// TIA Portal V17 export
// export: Created 2023-04-05T15:02:24.3314594Z, ExportSetting WithDefaults, DisplayName Totally Integrated Automation Portal, DisplayVersion V17 Update 4, DisplayName TIA Portal Openness, DisplayVersion V17 Update 4, DisplayName TIA Portal Version Control Interface, DisplayVersion V17, DisplayName STEP 7 Professional, DisplayVersion V17 Update 4, DisplayName STEP 7 Safety, DisplayVersion V17, DisplayName WinCC Professional, DisplayVersion V17 Update 4
FUNCTION_BLOCK "Main_Safety_RTG1"   // FB501, F_LAD
{ S7_Optimized_Access := 'TRUE' }
VERSION : 0.1
// stored: AutoNumber false, IsIECCheckEnabled false, UDAEnableTagReadback false
BEGIN

REGION Network 1: Receive data from Core - new
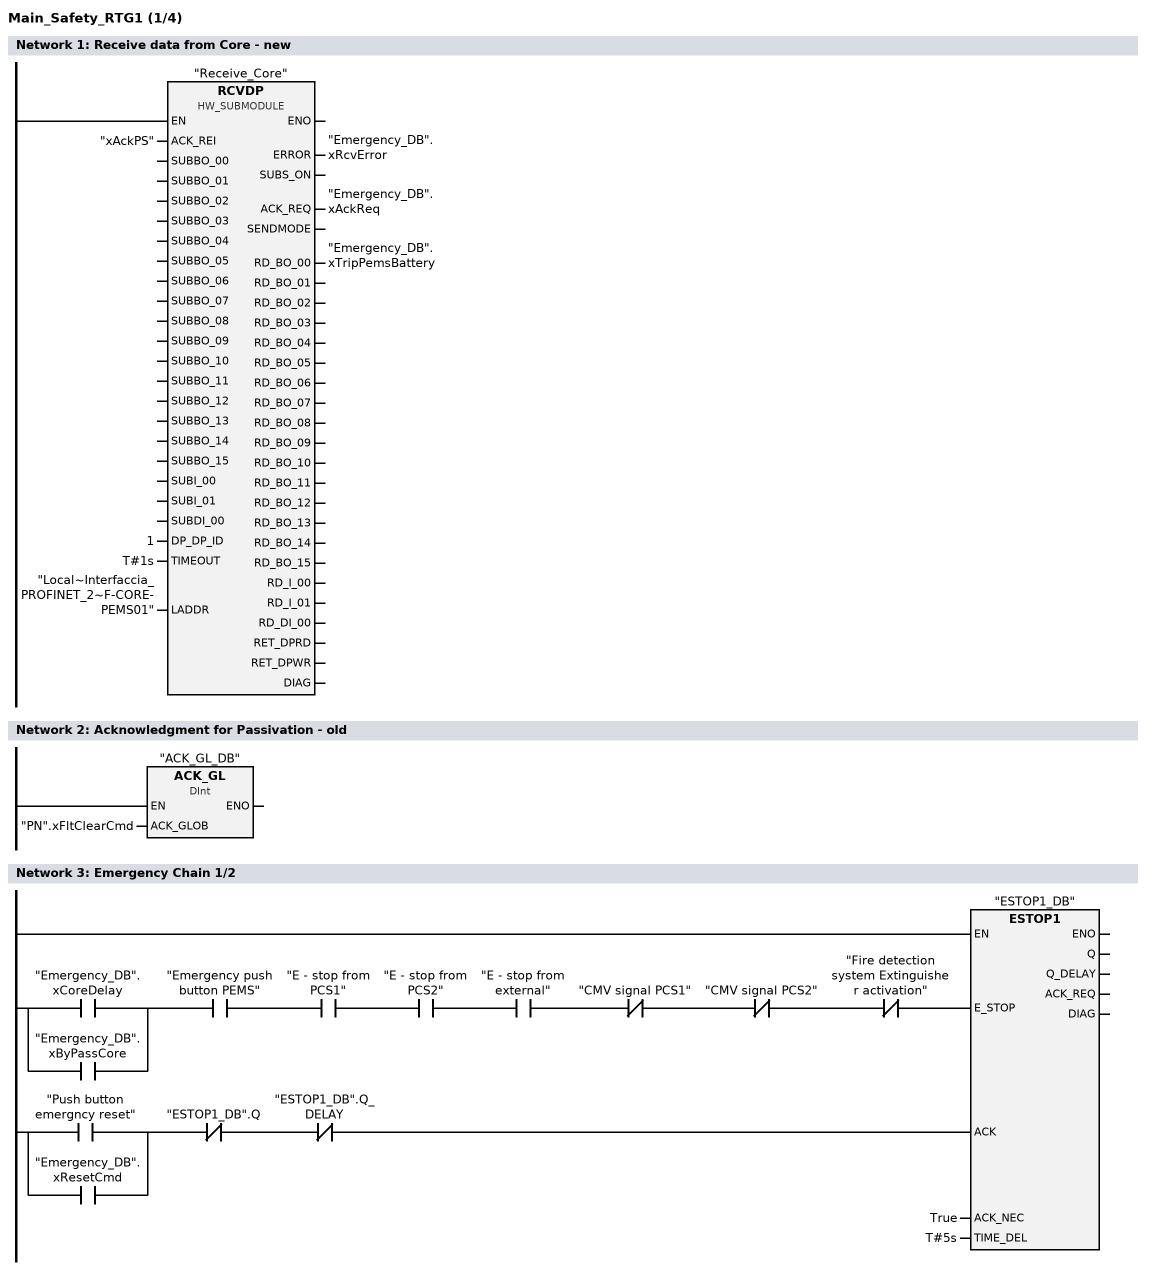
   RUNG wire#powerrail
      { S7_Templates := "laddr_type := HW_SUBMODULE" } "Receive_Core".RCVDP(ACK_REI := "xAckPS", SUBBO_00 :=, SUBBO_01 :=, SUBBO_02 :=, SUBBO_03 :=, SUBBO_04 :=, SUBBO_05 :=, SUBBO_06 :=, SUBBO_07 :=, SUBBO_08 :=, SUBBO_09 :=, SUBBO_10 :=, SUBBO_11 :=, SUBBO_12 :=, SUBBO_13 :=, SUBBO_14 :=, SUBBO_15 :=, SUBI_00 :=, SUBI_01 :=, SUBDI_00 :=, DP_DP_ID := 1, TIMEOUT := T#1s, LADDR := "Local~Interfaccia_PROFINET_2~F-CORE-PEMS01", ERROR => "Emergency_DB".xRcvError, SUBS_ON =>, ACK_REQ => "Emergency_DB".xAckReq, SENDMODE =>, RD_BO_00 => "Emergency_DB".xTripPemsBattery, RD_BO_01 =>, RD_BO_02 =>, RD_BO_03 =>, RD_BO_04 =>, RD_BO_05 =>, RD_BO_06 =>, RD_BO_07 =>, RD_BO_08 =>, RD_BO_09 =>, RD_BO_10 =>, RD_BO_11 =>, RD_BO_12 =>, RD_BO_13 =>, RD_BO_14 =>, RD_BO_15 =>, RD_I_00 =>, RD_I_01 =>, RD_DI_00 =>, RET_DPRD =>, RET_DPWR =>, DIAG =>)
   END_RUNG
   // the same network as SCL:
   "Receive_Core"(ACK_REI := "xAckPS",   // RCVDP
                  DP_DP_ID := 1,
                  TIMEOUT := T#1s,
                  LADDR := "Local~Interfaccia_PROFINET_2~F-CORE-PEMS01",
                  ERROR => "Emergency_DB".xRcvError,
                  ACK_REQ => "Emergency_DB".xAckReq,
                  RD_BO_00 => "Emergency_DB".xTripPemsBattery);
END_REGION

REGION Network 2: Acknowledgment for Passivation - old
   RUNG wire#powerrail
      { S7_Templates := "codedbool_type := DInt" } "ACK_GL_DB".ACK_GL(ACK_GLOB := "PN".xFltClearCmd)
   END_RUNG
   // the same network as SCL:
   "ACK_GL_DB"(ACK_GLOB := "PN".xFltClearCmd);   // ACK_GL
END_REGION

REGION Network 3: Emergency Chain 1/2
   RUNG wire#powerrail
      "ESTOP1_DB".ESTOP1(E_STOP := wire#w2, ACK := wire#w4, ACK_NEC := True, TIME_DEL := T#5s, Q =>, Q_DELAY =>, ACK_REQ =>, DIAG =>)
   END_RUNG
   RUNG wire#powerrail
      Contact( "Emergency_DB".xCoreDelay )
      wire#w1
      Contact( "Emergency push button PEMS" )
      Contact( "E - stop from PCS1" )
      Contact( "E - stop from PCS2" )
      Contact( "E - stop from external" )
      I_Contact( "CMV signal PCS1" )
      I_Contact( "CMV signal PCS2" )
      I_Contact( "Fire detection system Extinguisher activation" )
   END_RUNG wire#w2
   RUNG wire#powerrail
      Contact( "Emergency_DB".xByPassCore )
   END_RUNG wire#w1
   RUNG wire#powerrail
      Contact( "Push button emergncy reset" )
      wire#w3
      I_Contact( "ESTOP1_DB".Q )
      I_Contact( "ESTOP1_DB".Q_DELAY )
   END_RUNG wire#w4
   RUNG wire#powerrail
      Contact( "Emergency_DB".xResetCmd )
   END_RUNG wire#w3
   // the same network as SCL:
   "ESTOP1_DB"(E_STOP := ("Emergency_DB".xCoreDelay OR "Emergency_DB".xByPassCore) AND "Emergency push button PEMS" AND "E - stop from PCS1" AND "E - stop from PCS2" AND "E - stop from external" AND NOT "CMV signal PCS1" AND NOT "CMV signal PCS2" AND NOT "Fire detection system Extinguisher activation",   // ESTOP1
               ACK := ("Push button emergncy reset" OR "Emergency_DB".xResetCmd) AND NOT "ESTOP1_DB".Q AND NOT "ESTOP1_DB".Q_DELAY,
               ACK_NEC := True,
               TIME_DEL := T#5s);
END_REGION

REGION Network 4: Emergency shunt opening release RESET
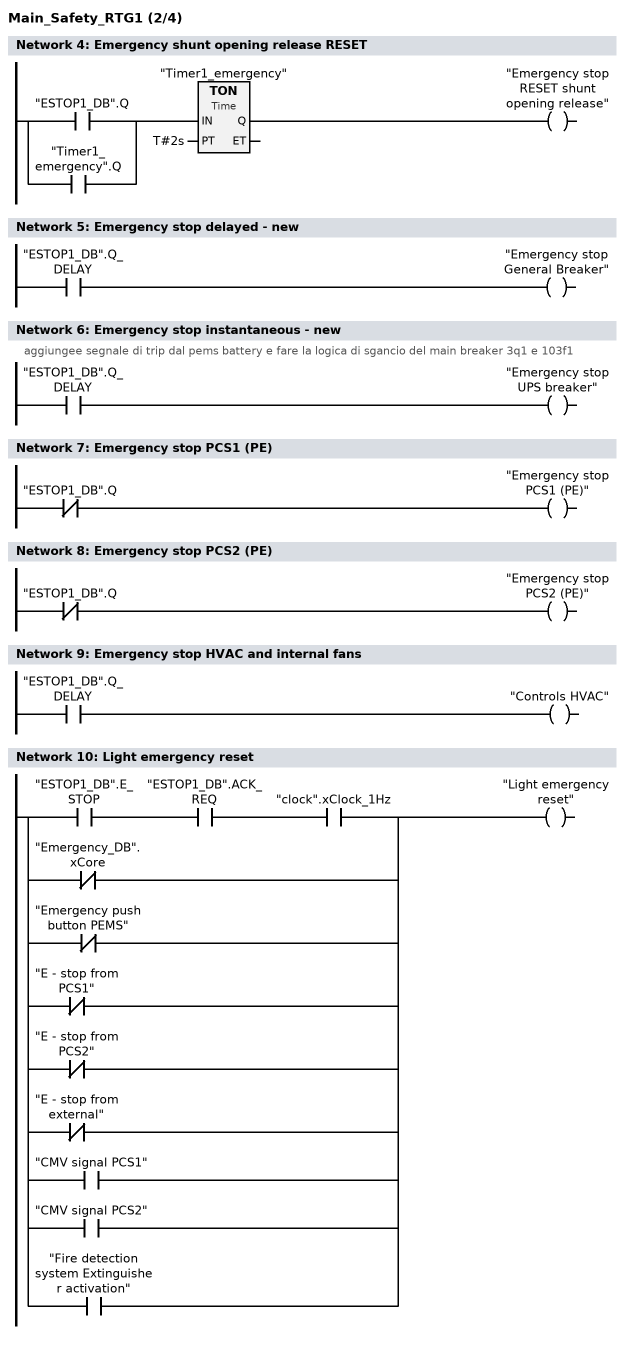
   RUNG wire#powerrail
      Contact( "ESTOP1_DB".Q )
      wire#w1
      { S7_Templates := "[time_type := Time, codedbool_type := DInt]" } "Timer1_emergency".TON(pt := T#2s, et =>)
      Coil( "Emergency stop RESET shunt opening release" )
   END_RUNG
   RUNG wire#powerrail
      Contact( "Timer1_emergency".Q )
   END_RUNG wire#w1
   // the same network as SCL:
   "Timer1_emergency".TON(IN := "ESTOP1_DB".Q OR "Timer1_emergency".Q, PT := T#2s);
   "Emergency stop RESET shunt opening release" := "Timer1_emergency".Q;
END_REGION

REGION Network 5: Emergency stop delayed - new
   RUNG wire#powerrail
      Contact( "ESTOP1_DB".Q_DELAY )
      Coil( "Emergency stop General Breaker" )
   END_RUNG
   // the same network as SCL:
   "Emergency stop General Breaker" := "ESTOP1_DB".Q_DELAY;
END_REGION

REGION Network 6: Emergency stop instantaneous - new
   // aggiungee segnale di trip dal pems battery e fare la logica di sgancio del main breaker 3q1 e 103f1
   RUNG wire#powerrail
      Contact( "ESTOP1_DB".Q_DELAY )
      Coil( "Emergency stop UPS breaker" )
   END_RUNG
   // the same network as SCL:
   "Emergency stop UPS breaker" := "ESTOP1_DB".Q_DELAY;
END_REGION

REGION Network 7: Emergency stop PCS1 (PE)
   RUNG wire#powerrail
      I_Contact( "ESTOP1_DB".Q )
      Coil( "Emergency stop PCS1 (PE)" )
   END_RUNG
   // the same network as SCL:
   "Emergency stop PCS1 (PE)" := NOT "ESTOP1_DB".Q;
END_REGION

REGION Network 8: Emergency stop PCS2 (PE)
   RUNG wire#powerrail
      I_Contact( "ESTOP1_DB".Q )
      Coil( "Emergency stop PCS2 (PE)" )
   END_RUNG
   // the same network as SCL:
   "Emergency stop PCS2 (PE)" := NOT "ESTOP1_DB".Q;
END_REGION

REGION Network 9: Emergency stop HVAC and internal fans
   RUNG wire#powerrail
      Contact( "ESTOP1_DB".Q_DELAY )
      Coil( "Controls HVAC" )
   END_RUNG
   // the same network as SCL:
   "Controls HVAC" := "ESTOP1_DB".Q_DELAY;
END_REGION

REGION Network 10: Light emergency reset
   RUNG wire#powerrail
      Contact( "ESTOP1_DB".E_STOP )
      Contact( "ESTOP1_DB".ACK_REQ )
      Contact( "clock".xClock_1Hz )
      wire#w1
      Coil( "Light emergency reset" )
   END_RUNG
   RUNG wire#powerrail
      I_Contact( "Emergency_DB".xCore )
   END_RUNG wire#w1
   RUNG wire#powerrail
      I_Contact( "Emergency push button PEMS" )
   END_RUNG wire#w1
   RUNG wire#powerrail
      I_Contact( "E - stop from PCS1" )
   END_RUNG wire#w1
   RUNG wire#powerrail
      I_Contact( "E - stop from PCS2" )
   END_RUNG wire#w1
   RUNG wire#powerrail
      I_Contact( "E - stop from external" )
   END_RUNG wire#w1
   RUNG wire#powerrail
      Contact( "CMV signal PCS1" )
   END_RUNG wire#w1
   RUNG wire#powerrail
      Contact( "CMV signal PCS2" )
   END_RUNG wire#w1
   RUNG wire#powerrail
      Contact( "Fire detection system Extinguisher activation" )
   END_RUNG wire#w1
   // the same network as SCL:
   "Light emergency reset" := ("ESTOP1_DB".E_STOP AND "ESTOP1_DB".ACK_REQ AND "clock".xClock_1Hz) OR NOT "Emergency_DB".xCore OR NOT "Emergency push button PEMS" OR NOT "E - stop from PCS1" OR NOT "E - stop from PCS2" OR NOT "E - stop from external" OR "CMV signal PCS1" OR "CMV signal PCS2" OR "Fire detection system Extinguisher activation";
END_REGION

REGION Network 11: Emergency - Open Battery Command
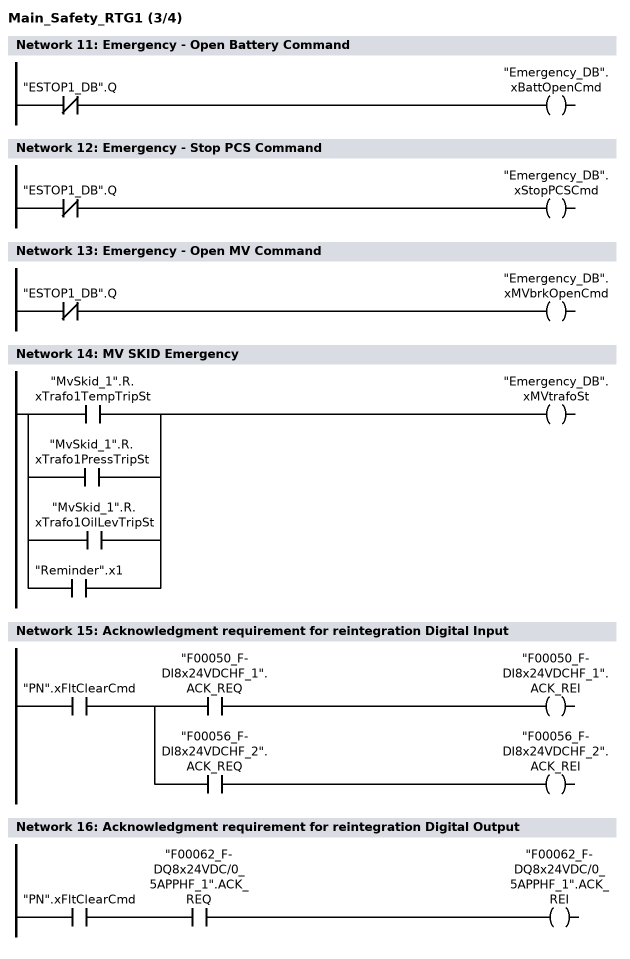
   RUNG wire#powerrail
      I_Contact( "ESTOP1_DB".Q )
      Coil( "Emergency_DB".xBattOpenCmd )
   END_RUNG
   // the same network as SCL:
   "Emergency_DB".xBattOpenCmd := NOT "ESTOP1_DB".Q;
END_REGION

REGION Network 12: Emergency - Stop PCS Command
   RUNG wire#powerrail
      I_Contact( "ESTOP1_DB".Q )
      Coil( "Emergency_DB".xStopPCSCmd )
   END_RUNG
   // the same network as SCL:
   "Emergency_DB".xStopPCSCmd := NOT "ESTOP1_DB".Q;
END_REGION

REGION Network 13: Emergency - Open MV Command
   RUNG wire#powerrail
      I_Contact( "ESTOP1_DB".Q )
      Coil( "Emergency_DB".xMVbrkOpenCmd )
   END_RUNG
   // the same network as SCL:
   "Emergency_DB".xMVbrkOpenCmd := NOT "ESTOP1_DB".Q;
END_REGION

REGION Network 14: MV SKID Emergency
   RUNG wire#powerrail
      Contact( "MvSkid_1".R.xTrafo1TempTripSt )
      wire#w1
      Coil( "Emergency_DB".xMVtrafoSt )
   END_RUNG
   RUNG wire#powerrail
      Contact( "MvSkid_1".R.xTrafo1PressTripSt )
   END_RUNG wire#w1
   RUNG wire#powerrail
      Contact( "MvSkid_1".R.xTrafo1OilLevTripSt )
   END_RUNG wire#w1
   RUNG wire#powerrail
      Contact( "Reminder".x1 )
   END_RUNG wire#w1
   // the same network as SCL:
   "Emergency_DB".xMVtrafoSt := "MvSkid_1".R.xTrafo1TempTripSt OR "MvSkid_1".R.xTrafo1PressTripSt OR "MvSkid_1".R.xTrafo1OilLevTripSt OR "Reminder".x1;
END_REGION

REGION Network 15: Acknowledgment requirement for reintegration Digital Input
   RUNG wire#powerrail
      Contact( "PN".xFltClearCmd )
      wire#w1
      Contact( "F00050_F-DI8x24VDCHF_1".ACK_REQ )
      Coil( "F00050_F-DI8x24VDCHF_1".ACK_REI )
   END_RUNG
   RUNG wire#w1
      Contact( "F00056_F-DI8x24VDCHF_2".ACK_REQ )
      Coil( "F00056_F-DI8x24VDCHF_2".ACK_REI )
   END_RUNG
   // the same network as SCL:
   "F00050_F-DI8x24VDCHF_1".ACK_REI := "PN".xFltClearCmd AND "F00050_F-DI8x24VDCHF_1".ACK_REQ;
   "F00056_F-DI8x24VDCHF_2".ACK_REI := "PN".xFltClearCmd AND "F00056_F-DI8x24VDCHF_2".ACK_REQ;
END_REGION

REGION Network 16: Acknowledgment requirement for reintegration Digital Output
   RUNG wire#powerrail
      Contact( "PN".xFltClearCmd )
      Contact( "F00062_F-DQ8x24VDC/0_5APPHF_1".ACK_REQ )
      Coil( "F00062_F-DQ8x24VDC/0_5APPHF_1".ACK_REI )
   END_RUNG
   // the same network as SCL:
   "F00062_F-DQ8x24VDC/0_5APPHF_1".ACK_REI := "PN".xFltClearCmd AND "F00062_F-DQ8x24VDC/0_5APPHF_1".ACK_REQ;
END_REGION

REGION Network 18: Send data to Core
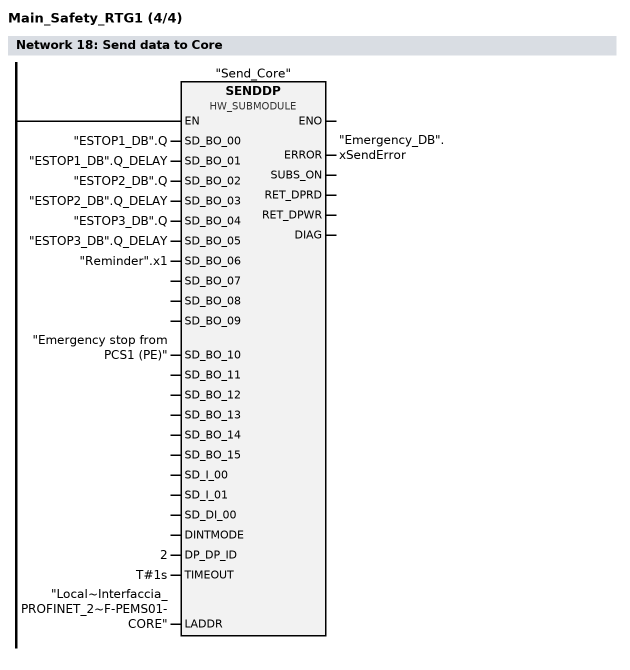
   RUNG wire#powerrail
      { S7_Templates := "laddr_type := HW_SUBMODULE" } "Send_Core".SENDDP(SD_BO_00 := "ESTOP1_DB".Q, SD_BO_01 := "ESTOP1_DB".Q_DELAY, SD_BO_02 := "ESTOP2_DB".Q, SD_BO_03 := "ESTOP2_DB".Q_DELAY, SD_BO_04 := "ESTOP3_DB".Q, SD_BO_05 := "ESTOP3_DB".Q_DELAY, SD_BO_06 := "Reminder".x1, SD_BO_07 :=, SD_BO_08 :=, SD_BO_09 :=, SD_BO_10 := "Emergency stop from PCS1 (PE)", SD_BO_11 :=, SD_BO_12 :=, SD_BO_13 :=, SD_BO_14 :=, SD_BO_15 :=, SD_I_00 :=, SD_I_01 :=, SD_DI_00 :=, DINTMODE :=, DP_DP_ID := 2, TIMEOUT := T#1s, LADDR := "Local~Interfaccia_PROFINET_2~F-PEMS01-CORE", ERROR => "Emergency_DB".xSendError, SUBS_ON =>, RET_DPRD =>, RET_DPWR =>, DIAG =>)
   END_RUNG
   // the same network as SCL:
   "Send_Core"(SD_BO_00 := "ESTOP1_DB".Q,   // SENDDP
               SD_BO_01 := "ESTOP1_DB".Q_DELAY,
               SD_BO_02 := "ESTOP2_DB".Q,
               SD_BO_03 := "ESTOP2_DB".Q_DELAY,
               SD_BO_04 := "ESTOP3_DB".Q,
               SD_BO_05 := "ESTOP3_DB".Q_DELAY,
               SD_BO_06 := "Reminder".x1,
               SD_BO_10 := "Emergency stop from PCS1 (PE)",
               DP_DP_ID := 2,
               TIMEOUT := T#1s,
               LADDR := "Local~Interfaccia_PROFINET_2~F-PEMS01-CORE",
               ERROR => "Emergency_DB".xSendError);
END_REGION
END_FUNCTION_BLOCK
